// Brief: Setup Arm Init
FUNCTION_BLOCK PUBLIC FB_SetupCtrlHold EXTENDS FB_SetupArmCtrlBase
VAR_INPUT
END_VAR
VAR_OUTPUT
END_VAR
VAR
	m_initState :INT :=0;
END_VAR

// override this function in each exact controller
METHOD PROTECTED calcCmdJntPos : BOOL
VAR_IN_OUT CONSTANT
	i_setupArm	:FB_SetupArm;
END_VAR


VAR 
	i :INT;
	curJntVel :Vec5d;
END_VAR
// set command joint position to current joint position, it's ok as all the joints is disabled.
// And by doing so, can avoid some fault triggers, like joint control error if joint enter disable too fast and brake can not stop joint immediately. 
IF m_timePeriod < 1.0 THEN
	m_cmdJntPos:=i_setupArm.curJntPos;
END_IF
END_METHOD

// override this function in each exact controller
// NOTICE: set joint control mode here, and do some initialization if needed
METHOD PUBLIC init : BOOL
VAR_IN_OUT CONSTANT
	i_setupArm	:FB_SetupArm;
END_VAR
VAR_IN_OUT 
	r_setupArmCtrlCmd :ST_SetupArmCtrlCmds;
END_VAR
SUPER^.Init(i_setupArm,r_setupArmCtrlCmd);

// TODO: setup joint3 would "jump" a bit when transit from torque mode to position mode
m_jntOPMode[3] := DriverOPMode_Trq;
END_METHOD

END_FUNCTION_BLOCK

(* stored: Version 1.1.0.1, ProductVersion 3.1.4024.11
   POU FB_SetupCtrlHold: Id {acc6ed82-034a-420c-8162-3225c33c4b38}, SpecialFunc None
   Method calcCmdJntPos: Id {0a1ec31f-6a67-4d62-bdf8-9fb476d6f874}
   Method init: Id {19914e93-fefd-4af6-8135-c232cbfbf440} *)
